FUNCTION_BLOCK FuseChannelBasic IMPLEMENTS IFuseChannelBasic
VAR_INPUT
END_VAR
VAR_OUTPUT
END_VAR
VAR
	_Chn : EL922x_ChannelBasic;
END_VAR


PROPERTY CoolDownLock : BOOL
GET
CoolDownLock := _Chn.Status.CoolDownLock;
END_GET
END_PROPERTY


PROPERTY CurrentLevelWarning : BOOL
GET
CurrentLevelWarning := _Chn.Status.CurrentLevelWarning;
END_GET
END_PROPERTY


PROPERTY Diag : BOOL
GET
Diag := _Chn.Status.Diag;
END_GET
END_PROPERTY


PROPERTY Enabled : BOOL
GET
Enabled := _Chn.Status.Enabled;
END_GET
END_PROPERTY


PROPERTY Error : BOOL
GET
Error := _Chn.Status.Error;
END_GET
END_PROPERTY


PROPERTY HardwareProtection : BOOL
GET
HardwareProtection := _Chn.Status.HWProtection;
END_GET
END_PROPERTY


METHOD ResetFuse : BOOL
_Chn.Control.Reset := NOT _Chn.Control.Reset;
END_METHOD


PROPERTY StateReset : BOOL
GET
StateReset := _Chn.Status.StateReset;
END_GET
END_PROPERTY


PROPERTY StateSwitch : BOOL
GET
StateSwitch := _Chn.Status.StateSwitch;
END_GET
END_PROPERTY

METHOD SwitchFuse : BOOL
_Chn.Control.Switch := NOT _Chn.Control.Switch;
END_METHOD


PROPERTY Tripped : BOOL
GET
Tripped := _Chn.Status.Tripped;
END_GET
END_PROPERTY


PROPERTY TxPDOState : BOOL
GET
TxPDOState := _Chn.Status.TxPDOState;
END_GET
END_PROPERTY

END_FUNCTION_BLOCK

(* stored: Version 1.1.0.1, ProductVersion 3.1.4024.6
   POU FuseChannelBasic: Id {d54f22cb-62e2-484b-a2d3-39cc584ea793}, SpecialFunc None
   Property CoolDownLock: Id {ce2f647a-40e5-469b-b1a8-ab6cdd4ef83b}
   Get Get: Id {07ab9f42-2eaa-4756-9a8b-a21903609f9e}
   Property CurrentLevelWarning: Id {733055b8-a014-436e-910e-c19d75f15312}
   Get Get: Id {e7a54a38-e723-4d63-b892-60c796392ca5}
   Property Diag: Id {af198614-c8e7-43d5-8256-2eb45569d607}
   Get Get: Id {ff61bbcf-2ad6-448b-90e9-89cc7c92a56a}
   Property Enabled: Id {afd86398-de34-427e-9feb-0712f5266325}
   Get Get: Id {8c14ddd4-9d1f-4bc8-9bda-d151dec9e176}
   Property Error: Id {b814054a-66aa-464e-bb78-697e7b864ab1}
   Get Get: Id {77305731-2c13-4f34-a5e1-91fd5764466a}
   Property HardwareProtection: Id {1a4abbe7-af31-4bbb-a692-d9ec14cfbe49}
   Get Get: Id {e2cfb2c8-4071-44ca-bdbc-4630236eb124}
   Method ResetFuse: Id {2adfb21e-387b-4e40-b7ec-5c377e84d804}
   Property StateReset: Id {2eaf1dbe-80ca-446d-9489-893b79426514}
   Get Get: Id {078e5e4d-980e-4334-b496-1b567d509f1d}
   Property StateSwitch: Id {a8e36af3-b3fe-4e88-b37b-0db9ff417d4b}
   Get Get: Id {ea637677-dd58-4d45-a2bd-e31e382ef2cc}
   Method SwitchFuse: Id {cbcaac99-468f-421a-9d94-6987dd01e5b3}
   Property Tripped: Id {dd417a43-8269-4a66-8f64-3e1c43f241d1}
   Get Get: Id {c9d14ced-676d-4023-9cea-b4463caf6e42}
   Property TxPDOState: Id {da352eef-1c3e-4929-88e8-92f054693d99}
   Get Get: Id {cf37f417-1b97-47b5-bacd-07a0543b8dc5} *)
